(* IEC 61131-3 sources: SIGMATEK-Jumag-Utils-Examples/typeManipulation/Class/splitDINT, 1 file *)

(* ---- splitDINT.st ---- *)
(*!
<Class
	Name               = "splitDINT"
	Revision           = "0.0"
	RealtimeTask       = "false"
	CyclicTask         = "true"
	DefCyclictime      = "10 ms"
	BackgroundTask     = "false"
	Sigmatek           = "false"
	OSInterface        = "false"
	HighPriority       = "false"
	Automatic          = "false"
	UpdateMode         = "Prescan"
	SharedCommandTable = "true"
	Objectsize         = "(284,120)">
	<Channels>
		<Server Name="ClassSvr" Visualized="false" Initialize="false" WriteProtected="true" Retentive="false"/>
		<Server Name="iInput" Visualized="false" Initialize="true" WriteProtected="false" Retentive="false"/>
		<Server Name="LSB" Visualized="false" Initialize="false" WriteProtected="true" Retentive="false"/>
		<Server Name="mid_LSB" Visualized="false" Initialize="false" WriteProtected="true" Retentive="false"/>
		<Server Name="mid_MSB" Visualized="false" Initialize="false" WriteProtected="true" Retentive="false"/>
		<Server Name="MSB" Visualized="false" Initialize="false" WriteProtected="true" Retentive="false"/>
	</Channels>
	<Dependencies>
		<Files>
			<File Path=".\Source\typeManipulation.c"/>
		</Files>
	</Dependencies>
</Class>
*)
splitDINT : CLASS
  //Servers:
	ClassSvr 	: SvrChCmd_DINT;
	iInput 	: SvrCh_DINT;
	MSB 	: SvrCh_DINT;
	mid_MSB 	: SvrCh_DINT;
	mid_LSB 	: SvrCh_DINT;
	LSB 	: SvrCh_DINT;
  //Clients:
  //Variables:
		mMSB : BSINT
		[
		];

		mLSB : BSINT
		[
		];

		mMidMSB : BSINT
		[
		];

		mMidLSB : BSINT
		[
		];

  //Functions:

	FUNCTION VIRTUAL GLOBAL CyWork
		VAR_INPUT
			EAX 	: UDINT;
		END_VAR
		VAR_OUTPUT
			state (EAX) 	: UDINT;
		END_VAR;
  //Tables:
	FUNCTION @STD
		VAR_OUTPUT
			ret_code	: CONFSTATES;
		END_VAR;
	FUNCTION GLOBAL TAB @CT_;
END_CLASS;

Function Global __cdecl splitDINT
VAR_INPUT
  IN : DINT;
  MSB : ^BSINT;
  MID_MSB : ^BSINT;
  MID_LSB : ^BSINT;
  LSB : ^BSINT;
END_VAR
VAR_OUTPUT
  Q : UINT;
END_VAR;

FUNCTION VIRTUAL GLOBAL splitDINT::CyWork
	VAR_INPUT
		EAX 	: UDINT;
	END_VAR
	VAR_OUTPUT
		state (EAX) 	: UDINT;
	END_VAR

  splitDINT(IN:=iInput, MSB:=#mMSB, MID_MSB:=#mMidMSB, MID_LSB:=#mMidLSB, LSB:=#mLSB);

  MSB := to_dint(mMSB);
  mid_MSB := to_dint(mMidMSB);
  mid_LSB := to_dint(mMidLSB);
  LSB := to_dint(mLSB);

	state := READY;

END_FUNCTION
